{attribute 'qualified_only'}
{attribute 'strict'}

TYPE STATI :
(
	S0 := 0, S1, S2, S3, SE, SA
);
END_TYPE

(* stored: Version 1.1.0.1, ProductVersion 3.1.4024.12
   EnumerationTextList DUT: Id {a829c61e-857d-48d5-8cce-fb6a46272340} *)
